(* IEC 61131-3 sources: LAxisCtrl/src/blocks, 1 file *)

(* ---- LAxisCtrl_AxisControl.st ---- *)
USING System.Math;
USING Siemens.Simatic.MotionControl.Native;

NAMESPACE Simatic.Ax.LAxisCtrl
    ///================================================================================
    /// SIEMENS AG
    /// (c)Copyright 2026 All Rights Reserved
    ///--------------------------------------------------------------------------------
    /// Library: LAxisCtrl
    /// Engineering: SIMATIC AX
    /// Restrictions: -
    /// Requirements: S7-1500T FW 4.0
    /// Functionality: This function block offers basic functionalities for axis control
    ///================================================================================
    FUNCTION_BLOCK AxisControl
        {S7.Extern = ReadWrite}
        VAR_INPUT
            /// TRUE: Enable functionality of FB
            enable : BOOL := FALSE;
            /// TRUE: Set axis enable; FALSE: Remove axis enable. MC_Power is used internally
            enableAxis : BOOL := FALSE;
            /// Rising edge: Acknowledgment of technology alarms or restart of the axis (depending on config). MC_Reset is used internally
            resetAxis : BOOL := FALSE;
            /// TRUE: Unconditionally open holding brake if axis is not enabled (e.g. for service purposes). Note: Do not modify this input while disabling of the axis is active (input enableAxis := FALSE and output axisEnabled = TRUE). MC_SetAxisSTW is used internally
            openBrake : BOOL := FALSE;
            /// Rising edge: Move an axis in jog mode (forward); Falling edge: Stop jogging. MC_MoveJog is used internally
            jogForward : BOOL := FALSE;
            /// Rising edge: Move an axis in jog mode (backward); Falling edge: Stop jogging. MC_MoveJog is used internally
            jogBackward : BOOL := FALSE;
            /// Rising edge: Move an axis at constant velocity/speed. MC_MoveVelocity is used internally
            moveVelocity : BOOL := FALSE;
            /// Rising edge: Brake an axis until it comes to a standstill. Note: MC_Halt is triggered internally
            stop : BOOL := FALSE;
            /// Rising edge: Brake an axis until it comes to a standstill (with fastStop dynamics). Note: MC_Halt is triggered internally
            fastStop : BOOL := FALSE;
            /// TRUE: Enable force/torque limiting. MC_TorqueLimiting is used internally
            torqueLimiting : BOOL := FALSE;
            /// Rising edge: Home axis. MC_Home is used internally
            homing : BOOL := FALSE;
            /// Rising edge: Move an axis relative to its position when execution of the job began. MC_MoveRelative is used internally
            posRelative : BOOL := FALSE;
            /// Rising edge: Move an axis to an absolute position. MC_MoveAbsolute is used internally
            posAbsolute : BOOL := FALSE;
            /// Rising edge: Start a superimposed positioning. MC_MoveSuperimposed is used internally
            posSuperimposed : BOOL := FALSE;
            /// Rising edge: Decelerate a superimposed motion to zero velocity. MC_HaltSuperimposed is used internally
            haltSuperimposed : BOOL := FALSE;
            /// Rising edge: Start a gearing operation (relative). MC_GearIn is used internally
            gearInRelative : BOOL := FALSE;
            /// Rising edge: Start a gearing operation (absolute). MC_GearInPos is used internally
            gearInAbsolute : BOOL := FALSE;
            /// Rising edge: Start a gearing operation (velocity synchronous). MC_GearInVelocity is used internally
            gearInVelocity : BOOL := FALSE;
            /// Rising edge: End a gearing/camming operation. MC_GearOut/MC_CamOut is used internally
            gearOutCamOut : BOOL := FALSE;
            /// Rising edge: Start a camming operation. MC_CamIn is used internally
            camIn : BOOL := FALSE;
            /// Rising edge: Start a phasing operation. MC_PhasingRelative/MC_PhasingAbsolute is used internally
            phasing : BOOL := FALSE;
            /// Rising edge: Start an offset operation. MC_OffsetRelative/MC_OffsetAbsolute is used internally
            offset : BOOL := FALSE;
            /// Reference to axis technology object to be controlled
            axis : DB_ANY  := UINT#0;
            /// Reference to leading axis technology object for synchronous motion
            master : DB_ANY := UINT#0;
            /// Cam technology object
            cam : DB_ANY := UINT#0;
            /// Structure for parameters
            config : typeAxisConfig;
        END_VAR

        {S7.Extern = ReadOnly}
        VAR_OUTPUT
            /// TRUE: Valid set of output values available at the FB
            valid : BOOL := FALSE;
            /// TRUE: FB is working and new output values can be expected
            busy : BOOL := FALSE;
            /// TRUE: An error occurred while processing the FB
            error : BOOL := FALSE;
            /// Current status of FB (16#0000 - 16#7FFF: Status of the FB, 16#8000 - 16#FFFF: Error identification)
            status : AxisStatus;
            /// Text of current status of FB
            statusText : String[STATUS_TEXT_LENGTH] := STRING#'STATUS_NO_CALL';
            /// Status of internally called subfunctions (ErrorID of Motion Control instructions)
            subfunctionStatus : WORD;
            /// TRUE: The technology object is enabled. Motion commands can be executed
            axisEnabled : BOOL := FALSE;
            /// TRUE: Reset/Restart of the axis is active
            resetActive : BOOL := FALSE;
            /// TRUE: The selected basic motion command is being executed
            commandBusy : BOOL := FALSE;
            /// TRUE: The selected basic motion command has completed without error
            commandDone : BOOL := FALSE;
            /// TRUE: The selected basic motion command has been aborted
            commandAborted : BOOL := FALSE;
            /// TRUE: The setpoint velocity/speed was reached and will be maintained
            inVelocity : BOOL := FALSE;
            /// TRUE: The drive is operating at the force/torque limit
            inLimitation : BOOL := FALSE;
            /// TRUE: Homing command is being executed
            homingCommandBusy : BOOL := FALSE;
            /// TRUE: Homing command has completed without error
            homingCommandDone : BOOL := FALSE;
            /// TRUE: Homing command has been aborted
            homingCommandAborted : BOOL := FALSE;
            /// TRUE: The selected superimposed motion command is being executed
            superimposedBusy : BOOL := FALSE;
            /// TRUE: The selected superimposed motion command  has completed without error
            superimposedDone : BOOL := FALSE;
            /// TRUE: The selected superimposed motion command has been aborted
            superimposedAborted : BOOL := FALSE;
            /// TRUE: The selected superimposed motion is active
            superimposedStart : BOOL := FALSE;
            /// TRUE: The drive is kept at the fixed stop (clamping), the axis position is within the positioning tolerance
            inClamping : BOOL := FALSE;
            /// TRUE: The axis is synchronizing to the leading axis / desynchronizing from the leading axis (Note: signal is only valid for the currently selected synchronous functionality, see outputs 'gearInAbsoluteSelected', 'gearInVelocitySelected', 'gearOutCamOutSelected' or 'camInSelected')
            startSync : BOOL := FALSE;
            /// TRUE: The axis is synchronized to the leading axis (Note: signal is only valid for the currently selected synchronous functionality, see outputs 'gearInRelativeSelected', 'gearInAbsoluteSelected', 'gearInVelocitySelected' or 'camInSelected')
            inSync : BOOL := FALSE;
            /// TRUE: The end of the cam has been reached. The output is displayed for at least one call when the cam is used cyclically
            endOfProfile : BOOL := FALSE;
            /// TRUE: Synchronous operation is being simulated
            inSimulation : BOOL := FALSE;
            /// TRUE: Jogging is active
            jogSelected : BOOL := FALSE;
            /// TRUE: Moving with constant velocity/speed is active
            moveVelocitySelected : BOOL := FALSE;
            /// TRUE: Stopping is active
            stopSelected : BOOL := FALSE;
            /// TRUE: Stopping is active (with fastStop dynamics)
            fastStopSelected : BOOL := FALSE;
            /// TRUE: Force/Torque limiting is active
            torqueLimitingSelected : BOOL := FALSE;
            /// TRUE: Homing is active
            homingSelected : BOOL := FALSE;
            /// TRUE: Relative positioning is active
            posRelativeSelected : BOOL := FALSE;
            /// TRUE: Absolute positioning is active
            posAbsoluteSelected : BOOL := FALSE;
            /// TRUE: Superimposed positioning is active (See also outputs: superimposedBusy, superimposedDone, superimposedAborted)
            posSuperimposedSelected : BOOL := FALSE;
            /// TRUE: Superimposed halting is active (See also outputs: superimposedBusy, superimposedDone, superimposedAborted)
            haltSuperimposedSelected : BOOL := FALSE;
            /// TRUE: Relative gearing is active (See also outputs: commandBusy, commandDone, commandAborted, inSync)
            gearInRelativeSelected : BOOL := FALSE;
            /// TRUE: Absolute gearing is active (See also outputs: commandBusy, commandDone, commandAborted, startSync, inSync)
            gearInAbsoluteSelected : BOOL := FALSE;
            /// TRUE: Velocity gearing is active (See also outputs: commandBusy, commandDone, commandAborted, startSync, inSync)
            gearInVelocitySelected : BOOL := FALSE;
            /// TRUE: End a gearing/camming operation is active (See also outputs: commandBusy, commandDone, commandAborted, startSync)
            gearOutCamOutSelected : BOOL := FALSE;
            /// TRUE: Camming is active (See also outputs: commandBusy, commandDone, commandAborted, startSync, inSync)
            camInSelected : BOOL := FALSE;
            /// TRUE: Phasing is active (See also outputs: superimposedBusy, superimposedDone, superimposedAborted, superimposedStart)
            phasingSelected : BOOL := FALSE;
            /// TRUE: Offset is active (See also outputs: superimposedBusy, superimposedDone, superimposedAborted, superimposedStart)
            offsetSelected : BOOL := FALSE;
            /// Diagnostics structure
            diagnostics : typeDiagnostics;
        END_VAR

        VAR
            /// Old value of statStatus
            _statusOld : AxisStatus;
            /// Internal text of current status of FB
            _statusText : String[STATUS_TEXT_LENGTH] := STRING#'STATUS_NO_CALL';
            /// Error occurred that can only be solved by user; rising edge at enable input necessary
            _errorUserCleared : BOOL := FALSE;
            /// Error occurred that can be acknowledged by FB
            _errorAutoCleared : BOOL := FALSE;
            /// Internal variable for status
            _status : AxisStatus;
            /// Internal variable for subfunction status
            _subfunctionStatus : WORD := WORD#16#0000;
            /// Internal variable for diagnostics
            _diagnostics : typeDiagnostics;
            /// Old value of enable for edge detection
            _enableOld : BOOL := FALSE;
            /// State of FB (function block state machine)
            _state : SINT := AXIS_MOTION;
            /// TRUE: First cycle of reset command
            _firstCycleReset : BOOL := TRUE;
            /// Old value of MC_Power.error
            _powerErrorOld : BOOL := FALSE;
            /// State of reset command
            _resetState : INT := CMD_IDLE;
            /// TRUE: First cycle of error in reset command
            _firstCycleResetError : BOOL := FALSE;
            /// Variable for requested extended command (e.g. resetAxis, torquelimiting, homing)
            _extendedCommand : DWORD := CMD_NO_SELECTION;
            /// Old value of variable for requested extended command
            _extendedCommandOld : DWORD := CMD_NO_SELECTION;
            /// Old value of enableAxis for edge detection
            _enableAxisOld : BOOL := FALSE;
            /// Internal empty diagnostic structure
            _emptyDiagnostics : typeDiagnostics;
            /// Old value of variable for homing command input
            _homingOld : BOOL := FALSE;
            /// TRUE: First cycle in homing command
            _firstCycleHoming : BOOL := TRUE;
            /// Current selected passive homing mode
            _passiveHomingState : DINT := NO_HOMING_ACTIVE;
            /// Current state of execution of homing command
            _exeOfHoming : INT := CMD_BUSY;
            /// Variable for requested basic motion command
            _basicCommand : DWORD := CMD_NO_SELECTION;
            /// Old value of variable for requested basic motion command
            _basicCommandOld : DWORD := CMD_NO_SELECTION;
            /// State of selected basic motion command
            _basicMotionState : DINT := NO_SELECTION;
            /// State of execution of current state of basic motion
            _exeOfBasicMotion : INT := CMD_BUSY;
            /// TRUE: First cycle in respective state for basic motion functionality
            _firstCycleBasicMotion : BOOL := TRUE;
            /// TRUE: applicative error occurred (e.g. invalid direction configured)
            _applicativeBasicMotionError : BOOL := FALSE;
            /// Velocity change on the fly is active
            _velocityChangeOnTheFly : BOOL := FALSE;
            /// Internal variable for velocity
            _basicVelocity : LREAL := 0.0;
            /// Internal variable for acceleration
            _basicAcceleration : LREAL := 0.0;
            /// Internal variable for deceleration
            _basicDeceleration : LREAL := 0.0;
            /// Internal variable for jerk
            _basicJerk : LREAL := 0.0;
            /// TRUE: First cycle of done at fastStop
            _firstCycleDone : BOOL := FALSE;
            /// Current executed state for torquelimiting functionality
            _torqueLimitingState : SINT := NO_TORQUE_LIMITING_ACTIVE;
            /// TRUE: Error at Torquelimiting occurred last cycle
            _torqueLimitingErrorOld : BOOL := FALSE;
            /// Current selected jog mode
            _jogMode : DINT := JOG_MODE_CONTINUOUS;
            /// Internal variable for direction of rotation of the axis
            _direction : INT := SPECIFIED_DIR;
            /// Internal variable for stopOnError function
            _stopWithoutSignalization : BOOL;
            /// Brake is opened
            _brakeOpened : BOOL;
            /// Brake change active
            _brakeChangeActive : BOOL;
            /// Edge detection
            _openBrakeOld : BOOL;
            /// The specified value is used according to the selected "Mode".
            _homingPosition : LREAL := 0.0;
            /// Current subState of execution of homing functionality
            _homingSubState : SINT := HOMING_IDLE;
            /// Current subState of execution of jog incremental functionality
            _incJogSubState : SINT := INC_JOG_IDLE;
            /// Last stored axis position (for incremental jogging)
            _incJogStartPosition : LREAL := 0.0;
            /// Old value of direction of executing incremental jogging
            _incJogDirectionOld : INT := 0;
            /// Jog Incremental: distance of Increment (positive or negative)
            _increment : LREAL := 0.0;
            /// Jog Incremental: current distance to destination position
            _incJogDistance : LREAL := 0.0;
            /// TRUE: First cycle in incremental jogging state (detection of new increment)
            _resetIncJog : BOOL := TRUE;
            /// Internal variable for position
            _position : LREAL := 0.0;
            /// Position change on the fly is active
            _positionChangeOnTheFly : BOOL := FALSE;
            /// Current selected active homing mode
            _activeHomingState : DINT := NO_HOMING_ACTIVE;
            /// Variable for requested superimposed motion command
            _supImpCommand : DWORD := CMD_NO_SELECTION;
            /// Old value of variable for requested superimposed motion command
            _supImpCommandOld : DWORD := CMD_NO_SELECTION;
            /// Current selected superimposed motion functionality
            _supImpMotionState : DINT := NO_SELECTION;
            /// Current state of execution of superimposed basic motion
            _exeOfSupImpMotionState : INT := CMD_BUSY;
            /// TRUE: First cycle in positioning (superimposed) functionality
            _firstCycleSupImpMotion : BOOL := TRUE;
            /// Position setpoint (for posSuperimposed command)
            _supImpMotionPosition : LREAL := 0.0;
            /// TRUE: applicative error occurred (e.g. invalid direction configured)
            _applicativeSupImpMotionError : BOOL := FALSE;
            /// Ratio change on the fly is active
            _ratioChangeOnTheFly : BOOL := FALSE;
            /// Gear ratio numerator
            _ratioNumerator : DINT := 1;
            /// Gear ratio denominator
            _ratioDenominator : DINT := 1;
            /// Phase shift change on the fly is active
            _changePhaseShiftOnTheFly : BOOL := FALSE;
            /// Offset change on the fly is active
            _changeOffsetOnTheFly : BOOL := FALSE;
            /// Relative/Absolute master value shift
            _phaseShift : LREAL := 0.0;
            /// Indicates the type of phase shift (TRUE: The phase shift is taken over as an absolute value; FALSE: The phase shift is added to an existing offset)
            _phaseAbsolute : BOOL := TRUE;
            /// Indicates the type of offset shift (TRUE: The offset shift is taken over as an absolute value; FALSE: The offset shift is added to an existing offset)
            _offsetAbsolute : BOOL := FALSE;
            /// Relative/Absolute offset
            _offsetValue : LREAL := 0.0;
            /// Type of axis
            _typeAxis : INT;
            /// Internal variable for enabling axis
            _enableAxis : BOOL := FALSE;
            /// Current executed state for synchronized motion simulation
            _syncMotionSimulationState : SINT := AXIS_NOT_IN_SIM;
            /// Old value of MC_SynchronizedMotionSimulation.error
            _synchronizedMotionErrorOld : BOOL := FALSE;
            /// Current executed State for execution of basic motion commands or reset of waiting gearing / camming commands
            _mainSelectionState : INT := 0;
            /// Application of cam
            _applicationMode : DINT := 0;
            /// Internal variable for waiting function state
            _waitingFunctionState : DINT := 0;
            /// Internal variable for waiting function state
            _waitingFunctionStateAbortAutomatic : DINT := -1;
            /// Internal variable for function state
            _functionState : DINT := 0;
            /// Internal variable
            _gearAndCamOutMode : DINT := 0;
            /// Internal variable
            _syncOutState : DINT;
            /// Internal old value for cam
            _camOld : DB_ANY;
            /// Internal old value for master
            _masterOld : DB_ANY;
            /// Internal reference of the technology object type TO_CamBase
            _refCamBase : REF_TO TO_CamBase;
            /// Internal reference of the technology object type TO_Axis (for the master axis)
            _refMasterAxis : REF_TO TO_Axis;
            /// Internal reference of the technology object type TO_Axis
            _refAxis : REF_TO TO_Axis;
            /// Internal reference of the technology object type TO_ExternalEncoder
            _refExtEncoder : REF_TO TO_ExternalEncoder;
            /// Internal reference of the technology object type TO_SpeedAxis
            _refSpeedAxis : REF_TO TO_SpeedAxis;
            /// Internal reference of the technology object type TO_PositioningAxis
            _refPosAxis : REF_TO TO_PositioningAxis;
            /// Internal reference of the technology object type TO_SynchronousAxis
            _refSyncAxis : REF_TO TO_SynchronousAxis;
            /// Instance of MC_Power
            _instPower : MC_POWER;
            /// Instance of MC_Reset
            _instReset : MC_RESET;
            /// Instance of MC_Home
            _instHome : MC_HOME;
            /// Instance of MC_Halt
            _instHalt : MC_HALT;
            /// Instance of MC_MoveJog
            _instMoveJog : MC_MOVEJOG;
            /// Instance of MC_TorqueLimiting
            _instTorqueLimiting : MC_TORQUELIMITING;
            /// Instance of MC_MoveVelocity
            _instMoveVelocity : MC_MOVEVELOCITY;
            /// Instance of MC_SetAxisSTW
            _instSetAxisSTW : MC_SETAXISSTW;
            /// Instance of MC_MoveRelative
            _instMoveRelative : MC_MOVERELATIVE;
            /// Instance of MC_MoveAbsolute
            _instMoveAbsolute : MC_MOVEABSOLUTE;
            /// Instance of MC_MoveSuperimposed
            _instMoveSuperimposed : MC_MOVESUPERIMPOSED;
            /// Instance of MC_HaltSuperimposed
            _instHaltSuperimposed : MC_HALTSUPERIMPOSED;
            /// Instance of MC_GearIn
            _instGearIn : MC_GEARIN;
            /// Instance of MC_PhasingAbsolute
            _instPhasingAbsolute : MC_PHASINGABSOLUTE;
            /// Instance of MC_PhasingRelative
            _instPhasingRelative : MC_PHASINGRELATIVE;
            /// Instance of MC_OffsetAbsolute
            _instOffsetAbsolute : MC_OFFSETABSOLUTE;
            /// Instance of MC_OffsetRelative
            _instOffsetRelative : MC_OFFSETRELATIVE;
            /// Instance of MC_GearInPos
            _instGearInPos : MC_GEARINPOS;
            /// Instance of MC_GearInVelocity
            _instGearInVelocity : MC_GEARINVELOCITY;
            /// Instance of MC_GearOut
            _instGearOut : MC_GEAROUT;
            /// Instance of MC_CamIn
            _instCamIn : MC_CAMIN;
            /// Instance of MC_CamOut
            _instCamOut : MC_CAMOUT;
            /// Instance of MC_SynchronizedMotionSimulation
            _instSyncMotionSimulation : MC_SYNCHRONIZEDMOTIONSIMULATION;
        END_VAR

        VAR_TEMP
            // Temporary variable for enable FB
            tempEnable : BOOL;
            // Temporary variable for extended command
            tempNewExtendedCmd : DINT;
            // Temporary variable for enableAxis
            tempEnableAxis : BOOL;
            // Temporary variable for error in actual command
            tempErrorInCmd : BOOL;
            // Temporary DWord which indicates all rising edges of command word
            tempRisingCmd : DWORD;
            // TRUE: Stop or faststop selected in current cycle
            tempStopCmdSelected : BOOL;
            // Temporary variable for statusword of axis
            tempStatusWord : DWORD;
            // Temporary variable for open brake
            tempOpenBrake : BOOL;
            // Temporary DWord for evaluation of rising edges of basic command word
            tempDword : DWORD;
            // Temporary index
            tempIndex : INT;
            // Temporary counter for rising edges in command word
            tempCountRisEdges : USINT;
            // Temporary variable for basic motion command
            tempNewBasicMotionCmd : DINT;
            // TRUE: State change is active, stay in loop for one more cycle
            tempStateChangeActive : BOOL;
            // Temporary variable for superimposed motion command
            tempNewSupImpCmd : DINT;
            // Temporary DInt variable
            tempDInt : DINT;
            // Temporary LReal variable
            tempLReal : LREAL;
            // Temporary Bool variable
            tempBool : BOOL;
            // Temporary variable for homing command
            tempHoming : BOOL;
        END_VAR

        VAR CONSTANT
            // Axis type: External encoder
            EXTERNAL_ENCODER : INT := 1;
            // Axis type: Speed axis
            SPEED_AXIS : INT := 2;
            // Axis type: Positioning axis
            POS_AXIS : INT := 3;
            // Axis type: Synchronous axis
            SYNC_AXIS : INT := 4;
            // Length of status text
            STATUS_TEXT_LENGTH : INT := 39;
            // State of FB: MotionState, new commands are evaluated
            AXIS_MOTION : SINT := SINT#1;
            // State of FB: Error, falling edge at FB_ENABLE required
            FB_ERROR : SINT := SINT#5;
            // No command is selected
            CMD_NO_SELECTION : DWORD := DWORD#16#0000_0000;
            // State of basicMotion/superimposedMotion: No execution of a command
            NO_SELECTION : INT := 0;

            // State of FB: StoppingState, MC_HALT is executed, new commands are not evaluated
            AXIS_FAST_STOPPING : SINT := SINT#2;
            // State of FB: ErrorState: Selection if StopOnError must be executed (depending on config)
            AXIS_STOP_ON_ERROR_SELECTION : SINT := SINT#3;
            // State of FB: ErrorState: Execution of StopOnError
            AXIS_STOP_ON_ERROR_EXECUTION : SINT := SINT#4;

            // Jogmode continuous selected (MC_MOVEJOG)
            JOG_MODE_CONTINUOUS : INT := 0;

            // State of basicMotion: Execution of fast stop command
            FAST_STOP_SELECTED : INT := 1;
            // State of basicMotion: Execution of stop command
            STOP_SELECTED : INT := 2;
            // State of basicMotion: Execution of jog forward command
            JOG_FORWARD_SELECTED : INT := 4;
            // State of basicMotion: Execution of jog backward command
            JOG_BACKWARD_SELECTED : INT := 8;
            // State of basicMotion: Execution of jog command if forward and backward are selected
            JOG_FW_AND_BW_SELECTED : INT := 12;
            // State of basicMotion: Execution of move velocity command
            MOVE_VELOCITY_SELECTED : INT := 16;
            // State of basicMotion: Execution of active homing command
            ACTIVE_HOMING_SELECTED : INT := 1024;
            // State of basicMotion: Execution of position command (relative)
            POS_RELATIVE_SELECTED : INT := 32;
            // State of basicMotion: Execution of position command (absolute)
            POS_ABSOLUTE_SELECTED : INT := 64;
            // State of basicMotion: Execution of gearIn command
            GEAR_IN_RELATIVE_SELECTED : INT := 128;
            // State of basicMotion: Execution of gearInPos command
            GEAR_IN_ABSOLUTE_SELECTED : INT := 256;
            // State of basicMotion: Execution of gearInVelocity command
            GEAR_IN_VELOCITY_SELECTED : INT := 4096;
            // State of basicMotion: Execution of camIn command
            CAM_IN_SELECTED : INT := 512;
            // State of basicMotion: Execution of gear and camOut command
            GEAR_OUT_CAM_OUT_SELECTED : INT := 2048;
            // State of superimposedMotion: Execution of posSuperimposed command
            POS_SUPERIMPOSED_SELECTED : INT := 1;
            // State of superimposedMotion: Execution of haltSuperimposed command
            HALT_SUPERIMPOSED_SELECTED : INT := 8;
            // State of superimposedMotion: Execution of phasing command
            PHASING_SELECTED : INT := 2;
            // State of superimposedMotion: Execution of offset command
            OFFSET_SELECTED : INT := 4;

            // State of basicMotion command: No execution
            CMD_IDLE : INT := 0;
            // State of basicMotion command: Subsequent call
            CMD_BUSY : INT := 1;
            // State of basicMotion command: Finished with "DONE"
            CMD_DONE : INT := 2;
            // State of basicMotion command: Finished with "ABORTED"
            CMD_ABORTED : INT := 4;
            // State of basicMotion command: Finished with "ERROR"
            CMD_ERROR : INT := 8;
            // State of basicMotion command: Finished with other reason
            CMD_END_PROCESS : INT := 16;

            // State of torquelimiting command: Not enabled
            NO_TORQUE_LIMITING_ACTIVE : SINT := SINT#0;
            // State of torquelimiting command: Torquelimiting is active
            TORQUE_LIMITING_SELECTED : SINT := SINT#1;
            // State of torquelimiting command: Torquelimiting is disabling
            TORQUE_LIMITING_DISABLE : SINT := SINT#10;

            // First bitposition for detecting rising edges at basic motion command word
            BITPOSITION_BASIC_MOTION_CMD : SINT := SINT#4;
            // Last bitposition for detecting rising edges at command word
            BIT_POS_LAST : SINT := SINT#15;
            // The sign of the velocity specified at the "Velocity" parameter defines the direction of rotation.
            SPECIFIED_DIR : INT := 0;
            // Bit 12 in STW
            MASK_STW_BIT12 : WORD := WORD#16#1000;

            // State of homing command: No homing active
            NO_HOMING_ACTIVE : SINT := SINT#-10;
            // State of homing command: (Standard) homing with MC_HOME
            STANDARD_HOMING : SINT := SINT#-1;

            // First bitposition for detecting rising edges at superimposed motion command word
            BITPOSITION_SUPERIMPOSED_MOTION_CMD : SINT := SINT#0;

            // State of torquelimiting command: Homing on fixed stop is active
            FIXED_STOP_DETECTION_ACTIVE : SINT := SINT#2;
            // State of torquelimiting command: Homing on fixed stop is finished
            FIXED_STOP_DETECTION_FINISHED : SINT := SINT#3;
            // State of torquelimiting command: Error occurred at homing on fixed stop process, axis is in clamping
            FIXED_STOP_DETECTION_ERROR_IN_CLAMPING : SINT := SINT#5;
            // State of torquelimiting command: Error occurred at homing on fixed stop process, axis is not in clamping
            FIXED_STOP_DETECTION_ERROR_NOT_IN_CLAMPING : SINT := SINT#6;

            // State of homing command: Applicative homing on fixed stop process active
            HOMING_ON_FIXED_STOP : SINT := SINT#0;
            // State of homing command: Applicative homing on fixed stop with moving out of clamping process active
            HOMING_ON_FIXED_STOP_WITH_MOVING_OUT_OF_CLAMPING : SINT := SINT#1;
            // State of homing command: Applicative homing on fixed stop with moving to target position process active
            HOMING_ON_FIXED_STOP_WITH_MOVING_TO_TARGET_POSITION : SINT := SINT#2;

            // Scaling factor for moving out of clamping. 1.0 = positioning window
            DISTANCE_SCALING : LREAL := 1.05;
            // Fixed stop detection (Mode for MC_TORQUELIMITING)
            MODE_FIXED_STOP_DETECTION : INT := 1;
            // Positive/Forward direction of rotation
            FORWARD_DIR : INT := 1;
            // Negative/Backward direction of rotation
            BACKWARD_DIR : INT := 2;
            // Shortest path
            SHORTEST_WAY_DIR : INT := 3;
            // Direct homing (absolute). Parameter "position" at MC_HOME is effective
            DIRECT_HOMING : INT := 0;
            // Active homing. Parameter "position" at MC_HOME is effective
            ACTIVE_HOMING : INT := 3;
            // Active homing. The configured home position value in technology object is effective
            ACTIVE_HOMING_TO_DEF_VALUE : INT := 5;
            // Absolute encoder adjustment (absolute)
            ABSOLUTE_ENCODER_ADJUSTMENT : INT := 7;
            // Encodertype INCREMENTAL
            INCREMENTAL_ENCODER : INT := 0;

            // SubState of homing on fixed stop process: Idle
            HOMING_IDLE : SINT := SINT#0;
            // SubState of homing on fixed stop process: Detecting fixed stop
            HOMING_FIXED_STOP_DETECTION : SINT := SINT#1;
            // SubState of homing on fixed stop process: Homeprocess (MC_HOME)
            HOMING_PROCESS : SINT := SINT#2;
            // SubState of homing on fixed stop process: Positioning to homeposition
            HOMING_POSITION : SINT := SINT#3;

            // Substate of incremental jog process: Idle
            INC_JOG_IDLE : SINT := SINT#0;
            // Substate of incremental jog process: Start moving
            INC_JOG_START : SINT := SINT#1;
            // Substate of incremental jog process: Stop moving
            INC_JOG_STOP : SINT := SINT#3;

            // Jogmode incremental selected - start always with new increment when command is selected
            JOG_MODE_NEW_INCREMENT : INT := 1;
            // Jogmode incremental selected - continue with increment when command is selected again
            JOG_MODE_CONTINUE_INCREMENT : INT := 2;
            // Application of the cam: Once/not cyclic (MC_CAMIN)
            APPLICATION_MODE_ONCE : INT := 0;
            // State of MainSelectionState: Regular execution of basic motion commands
            CALL_BASIC_MOTION : INT := 0;
            // State of MainSelectionState: Reset of waiting synchronous commands
            ABORT_WAITING_GEARINPOS_OR_CAMIN : INT := 1;

            // Mode for MC_GearOut / MC_CamOut instruction
            CANCEL_ONLY_WAITING_GEARING_CAMMING : DINT := 5;
            // No operation active or waiting
            WFS_FS_NO_OPERATION : DINT := 0;
            // Function state / Waiting function state: GearIn
            WFS_FS_GEARIN : DINT := 1;
            // Function state / Waiting function state: GearInPos
            WFS_FS_GEARINPOS : DINT := 2;
            // Function state / Waiting function state: CamIn
            WFS_FS_CAMIN : DINT := 3;
            // Function state / Waiting function state: Gearout
            WFS_FS_GEAROUT : DINT := 4;
            // Function state / Waiting function state: CamOut
            WFS_FS_CAMOUT : DINT := 5;

            // GearOutCamOut mode: Automatic
            SYNCOUT_MODE_AUTOMATIC : DINT := -1;
            // GearOutCamOut mode: GearOut
            SYNCOUT_MODE_GEAROUT : DINT := 0;
            // GearOutCamOut mode: CamOut
            SYNCOUT_MODE_CAMOUT : DINT := 1;
            // Sync out state
            SYNCOUT_STATE_CHECK_WAITING : INT := 1;
            // Sync out state
            SYNCOUT_STATE_GEAROUT_WAITING_BUSY : INT := 2;
            // Sync out state
            SYNCOUT_STATE_CAMOUT_WAITING_BUSY : INT := 3;
            // Sync out state
            SYNCOUT_STATE_CHECK_ACTIVE : INT := 4;
            // Sync out state
            SYNCOUT_STATE_GEAROUT_ACTIVE_BUSY : INT := 5;
            // Sync out state
            SYNCOUT_STATE_CAMOUT_ACTIVE_BUSY : INT := 6;
            // Sync out state
            SYNCOUT_STATE_DONE : INT := 7;
            // Sync out state
            SYNCOUT_STATE_ABORTED : INT := 8;
            // Sync out state
            SYNCOUT_STATE_ERROR : INT := 9;

            // State of motionSimulation: Axis is not in simulation
            AXIS_NOT_IN_SIM : SINT := SINT#0;
            // State of motionSimulation: Setting axis in simulation
            AXIS_STATE_SET_SIM : SINT := SINT#1;
            // State of motionSimulation: Disable axis
            AXIS_DISABLE : SINT := SINT#2;
            // State of motionSimulation: Axis is in simulation
            AXIS_STATE_IN_SIM : SINT := SINT#3;
            // State of motionSimulation: Enable axis
            AXIS_ENABLE : SINT := SINT#4;
            // State of motionSimulation: Resetting axis simulation
            AXIS_STATE_RESET_SIM : SINT := SINT#5;
        END_VAR

        //----------------------------------------------------------------------------------------------
        // Enable / disable FB
        //----------------------------------------------------------------------------------------------
        tempEnable := enable; // Create temporary process image
        IF NOT tempEnable AND _enableOld THEN

            // Reset outputs
            // ==========================================================
            // Error and valid outputs are reset with falling edge of enable input
            error := FALSE;
            valid := FALSE;
            status := AxisStatus#STATUS_NO_CALL;
            statusText := STRING#'STATUS_NO_CALL';
            subfunctionStatus := WORD#16#0000;
            _subfunctionStatus := WORD#16#0000;

            // Reset status outputs
            axisEnabled := FALSE;
            resetActive := FALSE;

            // Reset outputs for homing commands
            homingCommandBusy := FALSE;
            homingCommandDone := FALSE;
            homingCommandAborted := FALSE;
            homingSelected := FALSE;
            // Reset outputs for torquelimiting command
            torqueLimitingSelected := FALSE;
            inLimitation := FALSE;

            // Reset outputs for basic motion commands
            commandDone := FALSE;
            commandBusy := FALSE;
            commandAborted := FALSE;
            inVelocity := FALSE;
            fastStopSelected := FALSE;
            stopSelected := FALSE;
            jogSelected := FALSE;
            moveVelocitySelected := FALSE;
            // Outputs for for up to LAxisCtrl_PosAxis
            posRelativeSelected := FALSE;
            posAbsoluteSelected := FALSE;
            inClamping := FALSE;

            // Reset outputs for superimposed motion commands
            superimposedBusy := FALSE;
            superimposedDone := FALSE;
            superimposedAborted := FALSE;
            superimposedStart := FALSE;
            posSuperimposedSelected := FALSE;
            haltSuperimposedSelected := FALSE;
            startSync := FALSE;
            inSync := FALSE;
            endOfProfile := FALSE;
            gearInRelativeSelected := FALSE;
            inSimulation := FALSE;
            gearInAbsoluteSelected := FALSE;
            gearInVelocitySelected := FALSE;
            phasingSelected := FALSE;
            offsetSelected := FALSE;
            camInSelected := FALSE;
            gearOutCamOutSelected := FALSE;

            // Reset internal variables
            // ==========================================================
            _errorUserCleared := FALSE;
            _errorAutoCleared := FALSE;
            _status := AxisStatus#STATUS_NO_CALL;
            _statusOld := AxisStatus#STATUS_NO_CALL;
            _diagnostics := _emptyDiagnostics;

            _state := AXIS_MOTION;
            _firstCycleReset := FALSE;
            _powerErrorOld := FALSE;
            _resetState := CMD_IDLE;
            _firstCycleResetError := FALSE;

            _extendedCommand := CMD_NO_SELECTION;
            _extendedCommandOld := CMD_NO_SELECTION;
            _enableAxisOld := FALSE;
            _homingOld := FALSE;
            _firstCycleHoming := FALSE;
            _passiveHomingState := NO_HOMING_ACTIVE;
            _exeOfHoming := CMD_BUSY;
            _basicCommand := CMD_NO_SELECTION;
            _basicCommandOld := CMD_NO_SELECTION;
            _basicMotionState := NO_SELECTION;
            _exeOfBasicMotion := CMD_BUSY;
            _firstCycleBasicMotion := FALSE;
            _applicativeBasicMotionError := FALSE;
            _velocityChangeOnTheFly := FALSE;
            _basicVelocity := 0.0;
            _basicAcceleration := 0.0;
            _basicDeceleration := 0.0;
            _basicJerk := 0.0;

            _firstCycleDone := FALSE;

            _torqueLimitingState := NO_TORQUE_LIMITING_ACTIVE;
            _torqueLimitingErrorOld := FALSE;
            _jogMode := JOG_MODE_CONTINUOUS;
            _direction := SPECIFIED_DIR;

            _homingPosition := 0.0;
            _homingSubState := HOMING_IDLE;
            _incJogSubState := INC_JOG_IDLE;
            _incJogStartPosition := 0.0;
            _incJogDirectionOld := 0;
            _increment := 0.0;
            _incJogDistance := 0.0;
            _resetIncJog := TRUE;
            _position := 0.0;
            _positionChangeOnTheFly := FALSE;

            _activeHomingState := NO_HOMING_ACTIVE;
            _supImpCommand := CMD_NO_SELECTION;
            _supImpCommandOld := CMD_NO_SELECTION;
            _supImpMotionState := NO_SELECTION;
            _exeOfSupImpMotionState := CMD_BUSY;
            _firstCycleSupImpMotion := FALSE;
            _supImpMotionPosition := 0.0;
            _applicativeSupImpMotionError := FALSE;
            _ratioChangeOnTheFly := FALSE;
            _ratioNumerator := 0;
            _ratioDenominator := 0;
            // Tags for synchronized motion simulation
            _changePhaseShiftOnTheFly := FALSE;
            _changeOffsetOnTheFly := FALSE;
            _phaseShift := 0.0;
            _offsetValue := 0.0;
            _phaseAbsolute := TRUE;
            _offsetAbsolute := TRUE;
            _enableAxis := FALSE;
            _syncMotionSimulationState := AXIS_NOT_IN_SIM;
            _synchronizedMotionErrorOld := FALSE;
            _mainSelectionState := 0;
            _applicationMode := 0;

            _waitingFunctionState := 0;
            _waitingFunctionStateAbortAutomatic := -1;
            _functionState := 0;
            // ===========================================================

            // Disable Axis
            IF (_instPower.Busy = TRUE) THEN
                _instPower(Axis := _refAxis^,
                           Enable := FALSE,
                           StartMode := config.power.startMode,
                           StopMode := config.power.stopMode);
                // Check if error occurred
                IF (_instPower.Error = TRUE) THEN
                    // Write only diagnostics if error occurred at falling edge of MC_POWER
                    diagnostics.status := AxisStatus#ERR_MC_POWER;
                    diagnostics.subfunctionStatus := _instPower.ErrorId;
                    diagnostics.basicMotionState := _basicMotionState;
                    diagnostics.superimposedMotionState := _supImpMotionState;
                END_IF;
            END_IF;

            // Reset old values for master and cam
            _masterOld := UINT#0;
            _camOld := UINT#0;

            // Set axis references to null when block is being disabled
            _refAxis := NULL;
            _refSpeedAxis := NULL;
            _refPosAxis := NULL;
            _refSyncAxis := NULL;
            _refExtEncoder := NULL;
            _refMasterAxis := NULL;
            _refCamBase := NULL;

            // Set old value of enable for edge detection and end execution
            _enableOld := tempEnable;
            RETURN;

        // Check if FB is enabled - first cycle
        ELSIF tempEnable AND NOT _enableOld THEN

            // Busy is set at rising edge of enable input
            busy := TRUE;
            status := AxisStatus#STATUS_FB_FIRST_CALL;
            statusText := STRING#'STATUS_FB_FIRST_CALL';
            // StatStatus will be written in next cycle
            _status := AxisStatus#STATUS_SUBSEQUENT_CALL;
            _statusText := STRING#'STATUS_SUBSEQUENT_CALL';

            // Reset error and diagnostics outputs
            _errorUserCleared := FALSE;
            _errorAutoCleared := FALSE;
            diagnostics := _emptyDiagnostics;
            _diagnostics := _emptyDiagnostics;

            // Copy inputs
            _extendedCommand.%X0 := resetAxis;
            _basicCommand.%X8 := gearInAbsolute;
            _basicCommand.%X12 := gearInVelocity;
            _basicCommand.%X9 := camIn;
            _basicCommand.%X11 := gearOutCamOut;
            _supImpCommand.%X1 := phasing;
            _supImpCommand.%X2 := offset;
            _basicCommand.%X7 := gearInRelative;
            _basicCommand.%X5 := posRelative;
            _basicCommand.%X6 := posAbsolute;
            _supImpCommand.%X0 := posSuperimposed;
            _supImpCommand.%X3 := haltSuperimposed;
            _supImpCommandOld := _supImpCommand;

            _basicCommand.%X0 := fastStop;
            _basicCommand.%X1 := stop;
            _basicCommand.%X2 := jogForward;
            _basicCommand.%X3 := jogBackward;
            _basicCommand.%X4 := moveVelocity;
            _basicCommandOld := _basicCommand;
            // Set old value of homing input
            _homingOld := homing;

            _extendedCommandOld := _extendedCommand;
            // Set old value of enable for edge detection and end execution
            _enableOld := tempEnable;

            // resolve reference for axis input as TO_Axis (basic type for all axes)
            _refAxis := AsAxisRef(axis);
            IF _refAxis = NULL THEN
                // Invalid axis
                error := TRUE;
                _errorUserCleared := TRUE;
                status := AxisStatus#ERR_INVALID_AXIS;
                statusText := STRING#'ERR_INVALID_AXIS';
                diagnostics.status := AxisStatus#ERR_INVALID_AXIS;
            END_IF;

            CASE GetType(axis) OF
                TO_Type#SynchronousAxis:
                    _typeAxis := SYNC_AXIS;

                    // attempt to resolve all inherited technology objects (TO_SpeedAxis, TO_PositioningAxis, TO_SynchronousAxis)
                    _refSpeedAxis := AsSpeedAxisRef(axis);
                    _refPosAxis := AsPositioningAxisRef(axis);
                    _refSyncAxis := AsSynchronousAxisRef(axis);

                    // TODO: generate other error for this case?
                    IF _refSpeedAxis = NULL OR _refPosAxis = NULL OR _refSyncAxis = NULL THEN
                        // Invalid axis
                        error := TRUE;
                        _errorUserCleared := TRUE;
                        status := AxisStatus#ERR_INVALID_AXIS;
                        statusText := STRING#'ERR_INVALID_AXIS';
                        diagnostics.status := AxisStatus#ERR_INVALID_AXIS;
                    END_IF;

                TO_Type#PositioningAxis:
                    _typeAxis := POS_AXIS;

                    // attempt to resolve all inherited technology objects (TO_SpeedAxis, TO_PositioningAxis)
                    _refSpeedAxis := AsSpeedAxisRef(axis);
                    _refPosAxis := AsPositioningAxisRef(axis);

                    // TODO: generate other error for this case?
                    IF _refSpeedAxis = NULL OR _refPosAxis = NULL THEN
                        // Invalid axis
                        error := TRUE;
                        _errorUserCleared := TRUE;
                        status := AxisStatus#ERR_INVALID_AXIS;
                        statusText := STRING#'ERR_INVALID_AXIS';
                        diagnostics.status := AxisStatus#ERR_INVALID_AXIS;
                    END_IF;

                TO_Type#SpeedAxis:
                    _typeAxis := SPEED_AXIS;

                    _refSpeedAxis := AsSpeedAxisRef(axis);

                    // TODO: generate other error for this case?
                    IF _refSpeedAxis = NULL THEN
                        // Invalid axis
                        error := TRUE;
                        _errorUserCleared := TRUE;
                        status := AxisStatus#ERR_INVALID_AXIS;
                        statusText := STRING#'ERR_INVALID_AXIS';
                        diagnostics.status := AxisStatus#ERR_INVALID_AXIS;
                    END_IF;

                TO_Type#ExternalEncoder:
                    _typeAxis := EXTERNAL_ENCODER;

                    _refExtEncoder := AsExternalEncoderRef(axis);

                    // TODO: generate other error for this case?
                    IF _refExtEncoder = NULL THEN
                        // Invalid axis
                        error := TRUE;
                        _errorUserCleared := TRUE;
                        status := AxisStatus#ERR_INVALID_AXIS;
                        statusText := STRING#'ERR_INVALID_AXIS';
                        diagnostics.status := AxisStatus#ERR_INVALID_AXIS;
                    END_IF;

                ELSE
                    // Invalid axis
                    error := TRUE;
                    _errorUserCleared := TRUE;
                    status := AxisStatus#ERR_INVALID_AXIS;
                    statusText := STRING#'ERR_INVALID_AXIS';
                    diagnostics.status := AxisStatus#ERR_INVALID_AXIS;
            END_CASE;
        RETURN;

        // Check if function block is disabled or UserClearedError is present
        ELSIF NOT tempEnable OR _errorUserCleared THEN

            IF (tempEnable = FALSE) THEN
                status := AxisStatus#STATUS_NO_CALL;
                statusText := STRING#'STATUS_NO_CALL';
            END_IF;

            // Disable Axis
            IF (_instPower.Busy = TRUE) THEN
                _instPower(Axis := _refAxis^,
                           Enable := FALSE,
                           StartMode := config.power.startMode,
                           StopMode := config.power.stopMode);
                // Check if error occurred
                IF (_instPower.Error = TRUE) THEN
                    diagnostics.status := AxisStatus#ERR_MC_POWER;
                    diagnostics.subfunctionStatus := _instPower.ErrorId;
                    diagnostics.basicMotionState := _basicMotionState;
                    diagnostics.superimposedMotionState := _supImpMotionState;
                END_IF;
            ELSE
                // Reset if torque limiting is busy and axis is disabled
                IF (_instTorqueLimiting.Busy = TRUE)
                    OR (_instSyncMotionSimulation.Busy = TRUE)
                THEN
                    _instTorqueLimiting(Axis := _refSpeedAxis^,
                                        Enable := FALSE);
                    // Disable synchronized motion simulation
                    _instSyncMotionSimulation(Slave := _refSyncAxis^,
                                              Enable := FALSE);
                ELSE
                    busy := FALSE;
                END_IF;
            END_IF;

            // Reset old values for master and cam
            _masterOld := UINT#0;
            _camOld := UINT#0;

            // Set axis references to null when block is being disabled
            _refAxis := NULL;
            _refSpeedAxis := NULL;
            _refPosAxis := NULL;
            _refSyncAxis := NULL;
            _refExtEncoder := NULL;
            _refMasterAxis := NULL;
            _refCamBase := NULL;

            _enableOld := tempEnable;
            RETURN;

        ELSE

            // Read status word of the axis cyclically (needed for MC_Power call)
            CASE _typeAxis OF // Axis type is determined (checked) when the FB is enabled
                SPEED_AXIS, POS_AXIS, SYNC_AXIS:
                    // Axis type is TO_SpeedAxis or TO_PositioningAxis or TO_SynchronousAxis
                    tempStatusWord := _refSpeedAxis^.StatusWord;

                EXTERNAL_ENCODER:
                    // Axis type is TO_ExternalEncoder
                    tempStatusWord := _refExtEncoder^.StatusWord;

                ELSE
                    // Invalid axis
                    tempStatusWord := DWORD#16#0000_0000;
            END_CASE;

            // Copy extended inputs
            _extendedCommand.%X0 := resetAxis;
            tempEnableAxis := enableAxis;
            _extendedCommand.%X1 := torqueLimiting;
            _basicCommand.%X0 := fastStop;
            _basicCommand.%X1 := stop;
            _basicCommand.%X2 := jogForward;
            _basicCommand.%X3 := jogBackward;
            _basicCommand.%X4 := moveVelocity;
            tempOpenBrake := openBrake;
            _basicCommand.%X5 := posRelative;
            _basicCommand.%X6 := posAbsolute;
            _supImpCommand.%X0 := posSuperimposed;
            _supImpCommand.%X3 := haltSuperimposed;
            tempHoming := homing;
            IF (tempHoming = TRUE) AND (_homingOld = FALSE) THEN
                // Rising edge on homing input
                _extendedCommand.%X2 := TRUE;
                IF FALSE
                    OR (config.homing.extendedMode = HOMING_ON_FIXED_STOP) // Extended Homing mode (active)
                    OR (config.homing.extendedMode = HOMING_ON_FIXED_STOP_WITH_MOVING_OUT_OF_CLAMPING)  // Extended Homing mode (active)
                    OR (config.homing.extendedMode = HOMING_ON_FIXED_STOP_WITH_MOVING_TO_TARGET_POSITION)
                    OR (config.homing.extendedMode = -1) AND ((config.homing.mode = ACTIVE_HOMING) OR (config.homing.mode = ACTIVE_HOMING_TO_DEF_VALUE)) // Extended Homing mode (active)
                THEN
                    // Active Homing selected
                    _basicCommand.%X10 := TRUE; // Cmd is BasicMotionCmd
                    _extendedCommand.%X2 := FALSE;
                    // ELSE
                    //   ; // Passive Homing selected
                    //   // Bit in extended cmd already written
                END_IF;

            ELSIF (tempHoming = FALSE) AND (_homingOld = TRUE) THEN
                // Falling edge on homing input
                _extendedCommand.%X2 := FALSE;
                _basicCommand.%X10 := FALSE;
                // ELSE
                //   ; // Do nothing - wait for rising / Falling edge
            END_IF;
            _basicCommand.%X7 := gearInRelative;
            _basicCommand.%X8 := gearInAbsolute;
            _basicCommand.%X12 := gearInVelocity;
            _basicCommand.%X9 := camIn;
            _basicCommand.%X11 := gearOutCamOut;
            _supImpCommand.%X1 := phasing;
            _supImpCommand.%X2 := offset;

            // Statemachine for synchronized motion simulation

            REPEAT
                tempStateChangeActive := FALSE;
                CASE _syncMotionSimulationState OF
                    AXIS_NOT_IN_SIM:
                        // Axis NOT in simulation
                        IF (config.power.syncMotionSimulation = TRUE) THEN
                            // SynchronizedMotionSimulation is set
                            IF (tempEnableAxis = FALSE) AND (_enableAxisOld = TRUE) THEN
                                // Falling edge at enableAxis --> set simulation
                                CASE config.power.syncMotionSimulationExtendedMode OF
                                    -1: // Automatic when axis is in synchronous operation
                                        IF tempStatusWord.%X22 THEN // Check if axis is in synchronous operation
                                            _syncMotionSimulationState := AXIS_STATE_SET_SIM;
                                            _enableAxis := TRUE;
                                            tempStateChangeActive := TRUE;
                                        ELSE
                                            _enableAxis := tempEnableAxis;
                                        END_IF;

                                    0: // Start always simulation
                                        _syncMotionSimulationState := AXIS_STATE_SET_SIM;
                                        _enableAxis := TRUE;
                                        tempStateChangeActive := TRUE;
                                ELSE
                                    _enableAxis := tempEnableAxis; // : disable axis anyway
                                    // Error - Invalid extended mode
                                    _status := AxisStatus#ERR_INVALID_SYNCHRONIZED_EXTENDED_MODE;
                                    _statusText := STRING#'ERR_INVALID_SYNCHRONIZED_EXTENDED_MODE';
                                    _errorAutoCleared := TRUE;
                                    _diagnostics.basicMotionState := _basicMotionState;
                                    _diagnostics.superimposedMotionState := _supImpMotionState;
                                    _diagnostics.subfunctionStatus := WORD#0000;
                                    _subfunctionStatus := AxisStatus#STATUS_NO_CALL;
                                END_CASE;
                            ELSE
                                // FALSE or rising edge at input enableAxis
                                _enableAxis := tempEnableAxis;
                            END_IF;
                        ELSE
                            // SynchronizedMotionSimulation not set
                            // MC_POWER is only controlled by enableAxis input
                            _enableAxis := tempEnableAxis;
                        END_IF;

                    AXIS_STATE_SET_SIM:
                        // Set the axis in simulation
                        //----------------------------------------------------------
                        // Enable SynchronizedMotionSimulation
                        _instSyncMotionSimulation(Slave := _refSyncAxis^,
                                                  Enable := TRUE);
                        //----------------------------------------------------------
                        IF (_instSyncMotionSimulation.InSimulation = TRUE) THEN
                            _enableAxis := FALSE;
                            // Axis in Simulation - Change state
                            _syncMotionSimulationState := AXIS_DISABLE;
                        ELSIF (_instSyncMotionSimulation.Error = TRUE) THEN
                            // Error occurred - Disable Axis immediately
                            _enableAxis := FALSE;
                            _syncMotionSimulationState := AXIS_STATE_RESET_SIM;
                        // ELSE
                            //   ; // Wait for Axis is in simulation
                        END_IF;

                    AXIS_DISABLE:
                        // Disable axis
                        //----------------------------------------------------------
                        // Enable SynchronizedMotionSimulation
                        _instSyncMotionSimulation(Slave := _refSyncAxis^,
                                                  Enable := TRUE);
                        //----------------------------------------------------------
                        IF (_instPower.Error = TRUE) THEN
                            _syncMotionSimulationState := AXIS_STATE_RESET_SIM;
                        ELSIF (_instPower.Status = FALSE) THEN
                            // Axis disabled
                            _syncMotionSimulationState := AXIS_STATE_IN_SIM;
                        // ELSE
                            //   ; // Wait for Axis is disabled
                        END_IF;

                    AXIS_STATE_IN_SIM:
                        // Axis is in simulation
                        //----------------------------------------------------------
                        // Enable SynchronizedMotionSimulation
                        _instSyncMotionSimulation(Slave := _refSyncAxis^,
                                                  Enable := TRUE);
                        //----------------------------------------------------------
                        IF (tempEnableAxis = TRUE) AND (_enableAxisOld = FALSE) THEN
                            // Rising edge at enableAxis --> reset simulation
                            _syncMotionSimulationState := AXIS_ENABLE;
                            _enableAxis := TRUE;
                            tempStateChangeActive := TRUE;
                        ELSIF (config.power.syncMotionSimulation = FALSE) THEN
                            // End of synchronizedMotionSimulation by config without starting Axis
                            _syncMotionSimulationState := AXIS_STATE_RESET_SIM;
                            tempStateChangeActive := TRUE;
                        // ELSE
                            //   ; // Wait for rising edge at enableAxis
                        END_IF;

                    AXIS_ENABLE:
                        // Enable Axis
                        //----------------------------------------------------------
                        // Enable SynchronizedMotionSimulation while axis is enabling
                        _instSyncMotionSimulation(Slave := _refSyncAxis^,
                                                  Enable := TRUE);
                        //----------------------------------------------------------

                        IF (tempEnableAxis = FALSE) AND (_enableAxisOld = TRUE) THEN
                            _syncMotionSimulationState := AXIS_STATE_RESET_SIM;
                            _enableAxis := FALSE;
                        ELSIF (tempStatusWord.%X0 = TRUE) OR (_instPower.Error = TRUE)
                        // Reset simulation if axis is enabled or MC_POWER.STATUS = FALSE (Axis Error)
                        THEN
                            // FALSE on enable input
                            _syncMotionSimulationState := AXIS_STATE_RESET_SIM;
                            tempStateChangeActive := TRUE;
                        // ELSE
                            //   ; // Wait for Axis is Enabled
                        END_IF;

                    AXIS_STATE_RESET_SIM:
                        // Reset the axis simulation
                        //----------------------------------------------------------
                        // Enable SynchronizedMotionSimulation
                        _instSyncMotionSimulation(Slave := _refSyncAxis^,
                                                Enable := FALSE);
                        //----------------------------------------------------------
                        IF (_instSyncMotionSimulation.InSimulation = FALSE) AND (_instSyncMotionSimulation.Busy = FALSE) THEN
                            // Axis simulation is disabled
                            _syncMotionSimulationState := AXIS_NOT_IN_SIM;
                        // ELSE
                            //   ; // Wait for axis simulation is disabled
                        END_IF;

                        IF (tempEnableAxis = FALSE) AND (_enableAxisOld = TRUE) THEN
                            _enableAxis := FALSE;
                        END_IF;
                ELSE
                    // Errorhandling
                    _status := AxisStatus#ERR_UNDEFINED_MOTION_SIMULATION_STATE;
                    _statusText := STRING#'ERR_UNDEFINED_MOTION_SIMULATION_STATE';
                    _errorUserCleared := TRUE;
                    _diagnostics.subfunctionStatus := WORD#0000;
                    _subfunctionStatus := AxisStatus#STATUS_NO_CALL;
                    _diagnostics.basicMotionState := _basicMotionState;
                    _diagnostics.superimposedMotionState := _supImpMotionState;
                    // Set error state
                    _state := FB_ERROR;
                END_CASE;
            UNTIL (tempStateChangeActive = FALSE)
            END_REPEAT;

            // Evaluation of MC_Command
            IF (_instSyncMotionSimulation.Error = TRUE) AND (_synchronizedMotionErrorOld = FALSE) THEN
                // Errorhandling - Set error only at rising edge
                _errorAutoCleared := TRUE;
                _status := AxisStatus#ERR_MC_SYNCHRONIZEDMOTIONSIMULATION;
                _statusText := STRING#'ERR_MC_SYNCHRONIZEDMOTIONSIMULATION';
                _diagnostics.basicMotionState := _basicMotionState;
                _diagnostics.superimposedMotionState := _supImpMotionState;
                _diagnostics.subfunctionStatus := _instSyncMotionSimulation.ErrorId;
                _subfunctionStatus := _instSyncMotionSimulation.ErrorId;
            ELSIF (_instSyncMotionSimulation.Error = FALSE) AND (_status = AxisStatus#ERR_MC_SYNCHRONIZEDMOTIONSIMULATION)
            THEN
                // Reset error if error gone at respective Status
                _errorAutoCleared := FALSE;
                _status := AxisStatus#STATUS_SUBSEQUENT_CALL;
                _statusText := STRING#'STATUS_SUBSEQUENT_CALL';
            END_IF;
            _synchronizedMotionErrorOld := _instSyncMotionSimulation.Error;
            tempEnableAxis := _enableAxis;

            // Enable and disable axis
            IF (config.power.externalMC_PowerCall = FALSE) THEN
                // Call MC_POWER
                // Do not call the MC_Power instance if the axis is successfully enabled -> Reduce the runtime of the LAxisCtrl block
                // Only call the instance if at least one of the following conditions is fulfilled
                IF ((tempEnableAxis = TRUE) AND ((_instPower.Busy = FALSE) OR (_instPower.Status = FALSE))) // "enable axis" is given and enabling via MC_Power is in progress
                    OR (tempStatusWord.%X0 = FALSE) // Axis is disabled
                    OR (tempEnableAxis = FALSE) // "Remove axis enable" is set
                    OR (_instPower.Error = TRUE) // An error occurred in Motion Control instruction "MC_Power"
                THEN // Call the MC_Power instance
                    _instPower(Axis := _refAxis^,
                               Enable := tempEnableAxis,
                               StartMode := config.power.startMode,
                               StopMode := config.power.stopMode);
                END_IF;

                // Set and Reset of Error
                IF (_instPower.Error = TRUE) AND
                    ((_status = AxisStatus#STATUS_SUBSEQUENT_CALL) OR (_powerErrorOld = FALSE))
                THEN
                    // Error is set at rising edge of MC_POWER.Error
                    // Errorhandling
                    _status := AxisStatus#ERR_MC_POWER;
                    _statusText := STRING#'ERR_MC_POWER';
                    _errorAutoCleared := TRUE;
                    _diagnostics.basicMotionState := _basicMotionState;
                    _diagnostics.superimposedMotionState := _supImpMotionState;
                    _diagnostics.subfunctionStatus := _instPower.ErrorId;
                    _subfunctionStatus := _instPower.ErrorId;

                ELSIF (_status = AxisStatus#ERR_MC_POWER) AND (_instPower.Error = FALSE)
                THEN
                    // Reset Error
                    _status := AxisStatus#STATUS_SUBSEQUENT_CALL;
                    _statusText := STRING#'STATUS_SUBSEQUENT_CALL';
                    _errorAutoCleared := FALSE;

                ELSIF (tempEnableAxis = TRUE) AND (_enableAxisOld = FALSE) THEN
                    // Reset Error
                    _status := AxisStatus#STATUS_SUBSEQUENT_CALL;
                    _statusText := STRING#'STATUS_SUBSEQUENT_CALL';
                    _errorAutoCleared := FALSE;
                    _diagnostics := _emptyDiagnostics;
                // ELSE
                    //   ; // Do nothing
                END_IF;
            END_IF;

            IF tempOpenBrake AND NOT _openBrakeOld THEN
                // Open
                _instSetAxisSTW(Axis := _refSpeedAxis^,
                                Execute := FALSE,
                                STW1 := MASK_STW_BIT12,
                                STW1BitMask := MASK_STW_BIT12);
                _brakeChangeActive := TRUE;
                _brakeOpened := TRUE;

            ELSIF NOT tempOpenBrake AND _openBrakeOld THEN
                // Close
                _instSetAxisSTW(Axis := _refSpeedAxis^,
                                Execute := FALSE,
                                STW1 := WORD#16#0000,
                                STW1BitMask := MASK_STW_BIT12);
                _brakeChangeActive := TRUE;
                _brakeOpened := FALSE;
            END_IF;

            IF _brakeChangeActive THEN
                // Call of MC command
                _instSetAxisSTW(Axis := _refSpeedAxis^,
                                Execute := TRUE);

                IF NOT _instSetAxisSTW.Busy THEN
                    _brakeChangeActive := FALSE;
                END_IF;
            END_IF;

            // Edge detection
            _openBrakeOld := tempOpenBrake;
        END_IF;

        //----------------------------------------------------------------------------------------------
        // Resolve TO reference of master and cam
        //----------------------------------------------------------------------------------------------
        // resolve reference for master input as TO_Axis (every synchronous operation needs at least a type of TO_Axis for its master input)
        IF master <> UINT#0 AND master <> _masterOld THEN
            _refMasterAxis := AsAxisRef(master);

            // TODO: generate other error for this case?
            IF _refMasterAxis = NULL THEN
                // Invalid axis
                error := TRUE;
                _errorUserCleared := TRUE;
                status := AxisStatus#ERR_INVALID_AXIS;
                statusText := STRING#'ERR_INVALID_AXIS';
                diagnostics.status := AxisStatus#ERR_INVALID_AXIS;
            END_IF;
        END_IF;

        _masterOld := master;

        // resolve reference for cam input as TO_CamBase (every cam operation needs at least a type of TO_CamBase for its cam input)
        IF cam <> UINT#0 AND cam <> _camOld THEN
            _refCamBase := AsCamBaseRef(cam);

            // TODO: generate other error for this case?
            IF _refCamBase = NULL THEN
                // Invalid axis
                error := TRUE;
                _errorUserCleared := TRUE;
                status := AxisStatus#ERR_INVALID_AXIS;
                statusText := STRING#'ERR_INVALID_AXIS';
                diagnostics.status := AxisStatus#ERR_INVALID_AXIS;
            END_IF;
        END_IF;

        _camOld := cam;

        //----------------------------------------------------------------------------------------------
        // FB Statemachine
        //----------------------------------------------------------------------------------------------
        CASE _state OF
            AXIS_MOTION:
                // Check command inputs
                IF (_extendedCommand = CMD_NO_SELECTION)
                    AND (_basicCommand = CMD_NO_SELECTION)
                    AND (_supImpCommand = CMD_NO_SELECTION)
                THEN
                    // Command is reset
                    IF (_instPower.Error = TRUE) THEN
                        // Errorhandling
                        _status := AxisStatus#ERR_MC_POWER;
                        _statusText := STRING#'ERR_MC_POWER';
                        _errorAutoCleared := TRUE;
                    ELSIF (_instSyncMotionSimulation.Error = TRUE) THEN
                        ; // Do nothing

                    ELSIF (_instTorqueLimiting.Error = TRUE) THEN
                        ; // Do not reset if torque limiting error is pending

                    ELSE
                        // Reset Error only if no Error at MC_POWER is present
                        _status := AxisStatus#STATUS_SUBSEQUENT_CALL;
                        _statusText := STRING#'STATUS_SUBSEQUENT_CALL';
                        _errorAutoCleared := FALSE;
                    END_IF;

                ELSIF (_extendedCommand = _extendedCommandOld)
                    AND (_basicCommand = _basicCommandOld)
                    AND (_supImpCommand = _supImpCommandOld)
                THEN
                    ; // No change at command - do nothing

                ELSE
                    // Command changed
                    tempNewExtendedCmd := NO_SELECTION;
                    tempNewBasicMotionCmd := NO_SELECTION;
                    tempNewSupImpCmd := NO_SELECTION;
                    tempErrorInCmd := FALSE;

                    // Check basic motion command
                    IF (_basicCommand = _basicCommandOld) THEN
                        ; // Do nothing
                    ELSE
                        // Evaluate rising edges for basic motion command word - all rising edges of basic command word saved in tempRisingBasicCmd
                        tempRisingCmd := ((_basicCommand XOR _basicCommandOld) AND _basicCommand);
                        tempCountRisEdges := USINT#0; // Initialize counter for rising edges
                        // Count rising edges in tempRisingBasicCmd
                        FOR tempIndex := BITPOSITION_BASIC_MOTION_CMD TO BIT_POS_LAST DO
                            tempDword := SHR(tempRisingCmd, TO_USINT(tempIndex));
                            // Check for rising edge
                            IF (tempDword.%X0 = TRUE) THEN
                                tempCountRisEdges := tempCountRisEdges + USINT#1; // Increment at rising edge
                            END_IF;
                        END_FOR;
                        IF (tempRisingCmd.%X2 = TRUE) OR (tempRisingCmd.%X3 = TRUE) THEN
                            tempCountRisEdges := tempCountRisEdges + USINT#1; // jogForward AND/OR jogBackward is standing for 1 Command/rising edge
                        END_IF;

                        // Check Basic motion command
                        IF (tempCountRisEdges = 1)
                            OR (tempRisingCmd.%X0 = TRUE) // fastStop selected
                            OR (tempRisingCmd.%X1 = TRUE) // Stop selected
                        THEN
                            // Valid basic motion command selected
                            IF (tempRisingCmd.%X0 = TRUE) THEN
                                // FastStop selected
                                _state := AXIS_FAST_STOPPING;
                                tempNewBasicMotionCmd := FAST_STOP_SELECTED;
                                tempStopCmdSelected := TRUE;
                            ELSIF (tempRisingCmd.%X1 = TRUE) THEN
                                // Stop selected
                                tempNewBasicMotionCmd := STOP_SELECTED;
                                tempStopCmdSelected := TRUE;
                            ELSE
                                // Valid basic command priority 3 selected
                                // Set basic motion state
                                tempNewBasicMotionCmd := TO_DINT(tempRisingCmd);
                            END_IF;

                        ELSIF (tempCountRisEdges > 1) THEN
                            // Errorhandling - Invalid command
                            _status := AxisStatus#ERR_INVALID_BASIC_MOTION_CMD;
                            _statusText := STRING#'ERR_INVALID_BASIC_MOTION_CMD';
                            tempErrorInCmd := TRUE;
                        // ELSE
                            //   ; // Falling edge detection
                        END_IF;
                    END_IF;

                    // Check superimposed motion command
                    IF (_supImpCommand = _supImpCommandOld) THEN
                        ; // Do nothing
                    ELSE
                        // Superimposed motion command selected
                        IF (tempErrorInCmd = FALSE) AND // No Stop command selected in current cycle
                            (tempStopCmdSelected = FALSE)
                        THEN
                            tempRisingCmd := ((_supImpCommand XOR _supImpCommandOld) AND _supImpCommand);
                            tempCountRisEdges := USINT#0; // Initialize counter for rising edges
                            // Count rising edges in tempRisingSupImpCmd
                            FOR tempIndex := BITPOSITION_SUPERIMPOSED_MOTION_CMD TO BIT_POS_LAST DO
                                tempDword := SHR(tempRisingCmd, TO_USINT(tempIndex));
                                // Check for rising edge
                                IF (tempDword.%X0 = TRUE) THEN
                                    tempCountRisEdges := tempCountRisEdges + USINT#1;
                                END_IF;
                            END_FOR;

                            IF (tempCountRisEdges = 1) THEN
                                // Valid superimposed motion command
                                tempNewSupImpCmd := TO_DINT(tempRisingCmd);

                            ELSIF (tempCountRisEdges > 1) THEN
                                // Invalid Superimposed motion command
                                _status := AxisStatus#ERR_INVALID_SUPERIMPOSED_MOTION_CMD;
                                _statusText := STRING#'ERR_INVALID_SUPERIMPOSED_MOTION_CMD';
                                tempErrorInCmd := TRUE;
                            // ELSE
                                //   ; // Falling edge detection
                            END_IF;
                        // ELSE
                            //   ; // Stop or Faststop command selected OR error in BasicCommand
                        END_IF;
                    END_IF;

                    // Check extended command (reset, homing, torquelimiting)
                    IF (_extendedCommand = _extendedCommandOld) THEN
                        ; // Do nothing
                    ELSE
                        // Extended command selected
                        IF (tempErrorInCmd = FALSE) THEN
                            tempRisingCmd := ((_extendedCommand XOR _extendedCommandOld) AND _extendedCommand);
                            // Rising edge on torquelimiting command
                            IF (tempRisingCmd.%X1 = TRUE) THEN
                                tempNewExtendedCmd.%X1 := TRUE;
                                // Rising Edge at Homing on Fixed Stop and Torquelimiting
                                IF (tempNewBasicMotionCmd.%X10 = TRUE) AND (config.homing.extendedMode = 0) THEN
                                    // Errorhandling
                                    _status := AxisStatus#ERR_INVALID_EXTENDED_CMD;
                                    _statusText := STRING#'ERR_INVALID_EXTENDED_CMD';
                                    tempErrorInCmd := TRUE;
                                    tempNewExtendedCmd.%X1 := FALSE;

                                ELSIF (_torqueLimitingState = FIXED_STOP_DETECTION_ACTIVE)
                                THEN
                                    // Torquelimiting rejected because MC_TorqueLimiting is used during homing on fixed stop functionality
                                    _status := AxisStatus#ERR_TORQUE_LIMITING_NOT_ALLOWED;
                                    _statusText := STRING#'ERR_TORQUE_LIMITING_NOT_ALLOWED';
                                    tempErrorInCmd := TRUE;
                                    tempNewExtendedCmd.%X1 := FALSE;
                                    // ELSE
                                    //   ; // Start torquelimiting functionality
                                END_IF;
                            END_IF;

                            // Rising edge on passive homing command
                            IF (tempRisingCmd.%X2 = TRUE) THEN
                                tempNewExtendedCmd.%X2 := TRUE;
                                IF TRUE
                                    AND (_basicMotionState = ACTIVE_HOMING_SELECTED)
                                    AND ((_activeHomingState = HOMING_ON_FIXED_STOP) OR (_activeHomingState = HOMING_ON_FIXED_STOP_WITH_MOVING_OUT_OF_CLAMPING) OR (_activeHomingState = HOMING_ON_FIXED_STOP_WITH_MOVING_TO_TARGET_POSITION))
                                    AND (_exeOfBasicMotion = CMD_BUSY)
                                THEN
                                    // Passive Homing selected at homing on fixed stop
                                    _status := AxisStatus#ERR_HOMING_MODE_NOT_ALLOWED;
                                    _statusText := STRING#'ERR_HOMING_MODE_NOT_ALLOWED';
                                    tempErrorInCmd := TRUE;
                                    tempNewExtendedCmd.%X2 := FALSE;
                                    // ELSE
                                    //   ; // No error occurred
                                END_IF;
                            END_IF;
                        ELSE
                            ; // Error in basic motion command or superimposed motion command
                        END_IF;
                    END_IF;

                    // Enable commands
                    IF (tempErrorInCmd = TRUE) AND (tempStopCmdSelected = FALSE) THEN
                        // Error in current command - No Execution
                        _errorAutoCleared := TRUE;
                        _diagnostics.subfunctionStatus := WORD#0000;
                        _subfunctionStatus := AxisStatus#STATUS_NO_CALL;
                        // Write diagnostics
                        _diagnostics.basicMotionState := _basicMotionState;
                        _diagnostics.superimposedMotionState := _supImpMotionState;
                        _resetIncJog := TRUE;
                        // Set next state
                        _state := AXIS_STOP_ON_ERROR_SELECTION;
                    ELSE
                        // No Error in command occurred
                        IF (
                            (tempNewExtendedCmd <> NO_SELECTION)
                            OR (tempNewBasicMotionCmd <> NO_SELECTION)
                            OR (tempNewSupImpCmd <> NO_SELECTION)
                            )
                            OR (tempStopCmdSelected = TRUE)
                        THEN

                            // New valid command selected
                            // Basic motion commands
                            IF (tempNewBasicMotionCmd <> NO_SELECTION) THEN
                                _mainSelectionState := CALL_BASIC_MOTION;

                                IF config.generalSettings.abortWaitingSyncCmd THEN
                                    // Get axis waiting function state
                                    IF (_typeAxis = SYNC_AXIS) THEN
                                        _waitingFunctionStateAbortAutomatic := _refSyncAxis^.StatusSynchronizedMotion.WaitingFunctionState;
                                    END_IF;

                                    CASE _waitingFunctionStateAbortAutomatic OF
                                        WFS_FS_GEARINPOS, // Waiting
                                        WFS_FS_CAMIN: // Waiting
                                            // Waiting sync command
                                            CASE tempNewBasicMotionCmd OF
                                                GEAR_IN_ABSOLUTE_SELECTED,
                                                GEAR_IN_VELOCITY_SELECTED,
                                                CAM_IN_SELECTED,
                                                GEAR_IN_RELATIVE_SELECTED,
                                                GEAR_OUT_CAM_OUT_SELECTED:
                                                    ; // New command aborts waiting sync command
                                            ELSE
                                                _mainSelectionState := ABORT_WAITING_GEARINPOS_OR_CAMIN; // Reset waiting absolute gearing / camIn command
                                            END_CASE;
                                    ELSE
                                        ;
                                    END_CASE;

                                    IF (_mainSelectionState = ABORT_WAITING_GEARINPOS_OR_CAMIN) THEN
                                        // Reset instance of MC_GearOut / MC_CamOut
                                        CASE _waitingFunctionStateAbortAutomatic OF
                                            WFS_FS_GEARINPOS: // Waiting
                                                _instGearOut(Slave := _refSyncAxis^,
                                                            Execute := FALSE,
                                                            SyncProfileReference := CANCEL_ONLY_WAITING_GEARING_CAMMING); // 5 = Abort waiting camming / gearing

                                            WFS_FS_CAMIN: // Waiting
                                                _instCamOut(Slave := _refSyncAxis^,
                                                            Execute := FALSE,
                                                            SyncProfileReference := CANCEL_ONLY_WAITING_GEARING_CAMMING); // 5 = Abort waiting camming / gearing
                                        END_CASE;
                                    END_IF;
                                ELSE
                                    // Automatic abort of waiting sync commands not enabled
                                    _waitingFunctionStateAbortAutomatic := -1;
                                END_IF;

                                _firstCycleBasicMotion := TRUE;
                                // Evaluate if Jog command is set
                                IF (tempNewBasicMotionCmd.%X2 = TRUE) OR (tempNewBasicMotionCmd.%X3 = TRUE) THEN
                                    _exeOfBasicMotion := CMD_BUSY;
                                    // Select Jogmode
                                    IF ((_basicCommand.%X2 = FALSE) AND (tempNewBasicMotionCmd.%X3 = TRUE)) OR // Rising edge at JogBackward and JogForward = FALSE
                                        ((_basicCommand.%X3 = FALSE) AND (tempNewBasicMotionCmd.%X2 = TRUE)) OR // Only rising edge at JogForward and JogBackward = FALSE
                                        ((tempNewBasicMotionCmd.%X2 = TRUE) AND (tempNewBasicMotionCmd.%X3 = TRUE)) // Rising edge at FW and BW
                                    THEN
                                        // One Input direction = False, other is rising edge, or both rising edge --> Start jog
                                        IF (_jogMode <> config.jog.mode) THEN
                                            _resetIncJog := TRUE;
                                        END_IF;
                                        _jogMode := config.jog.mode;
                                    ELSE
                                        // Rising edge at one input, the other is already TRUE - Dont Change Jogmode
                                        IF ((_basicMotionState = JOG_BACKWARD_SELECTED) OR (_basicMotionState = JOG_FORWARD_SELECTED)) AND (_jogMode <> JOG_MODE_CONTINUOUS)
                                        THEN
                                            _firstCycleBasicMotion := FALSE;
                                        END_IF;
                                    END_IF;
                                ELSE
                                    ; // Reset jog increment if other command than jog selected
                                    _resetIncJog := TRUE;
                                END_IF;

                                // Set new basic motion state
                                _basicMotionState := tempNewBasicMotionCmd;
                            END_IF;

                            // Superimposed motion commands
                            IF (tempNewSupImpCmd <> NO_SELECTION) THEN
                                _supImpMotionState := tempNewSupImpCmd;
                                _firstCycleSupImpMotion := TRUE;
                                _resetIncJog := TRUE;
                            END_IF;

                            // Extended commands

                            IF (tempNewExtendedCmd <> NO_SELECTION) THEN
                                IF (tempNewExtendedCmd.%X1 = TRUE) THEN
                                    // Rising edge on torquelimiting command
                                    IF (_torqueLimitingState = NO_TORQUE_LIMITING_ACTIVE) THEN
                                        // No torquelimiting active --> Enable torquelimiting
                                        _torqueLimitingState := TORQUE_LIMITING_SELECTED;
                                    END_IF;
                                END_IF;
                                // Homing command
                                IF (tempNewExtendedCmd.%X2 = TRUE) THEN
                                    _passiveHomingState := config.homing.extendedMode;
                                    _firstCycleHoming := TRUE;
                                    _resetIncJog := TRUE;
                                END_IF;
                            END_IF;

                        // Reset error
                        _status := AxisStatus#STATUS_SUBSEQUENT_CALL;
                        _statusText := STRING#'STATUS_SUBSEQUENT_CALL';
                        _errorAutoCleared := FALSE;
                        _diagnostics := _emptyDiagnostics;
                    // ELSE
                        //   ; // No rising edge at commands
                        END_IF;
                    END_IF;
                END_IF;

            AXIS_FAST_STOPPING:
                IF (config.fastStop.replaceStopPossible = FALSE) THEN
                    ; // Fast stop command can not be interrupted by another command
                    // State change is executed in FastStop implementation if command finished
                ELSE
                    _state := AXIS_MOTION;
                END_IF;

            AXIS_STOP_ON_ERROR_SELECTION,
            AXIS_STOP_ON_ERROR_EXECUTION:
                ; // Wait for stopping axis if StopOnError is configured
            FB_ERROR: // Error state
                ; // Do nothing, status already set

        ELSE
            // Errorhandling
            _status := AxisStatus#ERR_UNDEFINED_FB_STATE;
            _statusText := STRING#'ERR_UNDEFINED_FB_STATE';
            _errorUserCleared := TRUE;
            _diagnostics.subfunctionStatus := WORD#0000;
            _subfunctionStatus := AxisStatus#STATUS_NO_CALL;
            _diagnostics.basicMotionState := _basicMotionState;
            _diagnostics.superimposedMotionState := _supImpMotionState;
            // Set error state
            _state := FB_ERROR;
        END_CASE;

        //----------------------------------------------------------------------------------------------
        // Execution of reset functionality
        //----------------------------------------------------------------------------------------------

        // Firstcycle of command
        IF (_extendedCommand.%X0 = TRUE) AND (_extendedCommandOld.%X0 = FALSE) THEN
            _firstCycleReset := TRUE;
            // Reset MC_RESET command
            _instReset(Axis := _refAxis^,
                       Execute := FALSE,
                       Restart := config.generalSettings.resetWithRestart);
            _firstCycleResetError := FALSE;
            _resetState := CMD_BUSY;
        END_IF;

        CASE _resetState OF
            CMD_IDLE:
                ; // Do nothing

            CMD_BUSY:
                // Call MC_Command
                _instReset(Axis := _refAxis^,
                           Execute := _extendedCommand.%X0);

                // Evaluate MC_Command
                IF (_instReset.Error = TRUE) THEN
                    // Errorhandling
                    IF (_firstCycleResetError = FALSE) THEN
                        _errorAutoCleared := TRUE;
                        _status := AxisStatus#ERR_MC_RESET;
                        _statusText := STRING#'ERR_MC_RESET';
                        _diagnostics.basicMotionState := _basicMotionState;
                        _diagnostics.superimposedMotionState := _supImpMotionState;
                        _diagnostics.subfunctionStatus := _instReset.ErrorId;
                        _subfunctionStatus := _instReset.ErrorId;
                        _firstCycleResetError := TRUE;
                        // Set next state
                        _resetState := CMD_IDLE;
                        IF (_state = AXIS_MOTION) THEN
                        // Set TO_STOP_ON_ERROR State only if the current state is TO_MOTION
                        _state := AXIS_STOP_ON_ERROR_SELECTION;
                        END_IF;
                    END_IF;

                ELSIF (_instReset.Busy = FALSE) THEN
                    // Set next state
                    _resetState := CMD_IDLE;
                // ELSE
                //   ; // Command selected
                END_IF;
        ELSE
            // Errorhandling
            _status := AxisStatus#ERR_UNDEFINED_RESET_STATE;
            _statusText := STRING#'ERR_UNDEFINED_RESET_STATE';
            _errorUserCleared := TRUE;
            _diagnostics.subfunctionStatus := WORD#0000;
            _subfunctionStatus := AxisStatus#STATUS_NO_CALL;
            _diagnostics.basicMotionState := _basicMotionState;
            _diagnostics.superimposedMotionState := _supImpMotionState;
        END_CASE;

        //----------------------------------------------------------------------------------------------
        // Execution of functionalities of basic coordinate system
        //----------------------------------------------------------------------------------------------

        // Write diagnostics
        _diagnostics.basicMotionState := _basicMotionState;
        _diagnostics.superimposedMotionState := _supImpMotionState;
        REPEAT
            tempStateChangeActive := FALSE;
            // Statemachine for main selection state
            CASE _mainSelectionState OF
                CALL_BASIC_MOTION:
                    CASE _basicMotionState OF
                        NO_SELECTION:
                            ; // No execution

                        FAST_STOP_SELECTED:
                            ; // Implementation at end of code

                        STOP_SELECTED:
                            // No additional features

                            // Firstcycle of command
                            IF (_firstCycleBasicMotion = TRUE) THEN
                                // Reset HALT command
                                _instHalt(Axis := _refSpeedAxis^,
                                          Execute := FALSE,
                                          Deceleration := config.stop.deceleration,
                                          AbortAcceleration := config.stop.abortAcceleration,
                                          Jerk := config.stop.jerk,
                                          Mode := config.stop.haltMode); // New input 'Mode' as of Motion Control V9.0
                            END_IF;

                            // Call MC_Command
                            _instHalt(Axis := _refSpeedAxis^,
                                      Execute := _basicCommand.%X1 OR _firstCycleBasicMotion);

                            // Evaluate MC_Command
                            IF (_instHalt.Busy = FALSE) AND
                                (_instHalt.Error = FALSE) AND
                                (_instHalt.Done = FALSE) AND
                                (_instHalt.CommandAborted = FALSE)
                            THEN
                                // Return to NO_SELECTION if command finished
                                _basicMotionState := NO_SELECTION;

                            ELSIF (_instHalt.Error = TRUE) THEN
                                // Errorhandling
                                _status := AxisStatus#ERR_MC_HALT;
                                _statusText := STRING#'ERR_MC_HALT';
                                _errorAutoCleared := TRUE;
                                _diagnostics.subfunctionStatus := _instHalt.ErrorId;
                                _subfunctionStatus := _instHalt.ErrorId;
                                // Set next state
                                _state := AXIS_STOP_ON_ERROR_SELECTION;
                                _basicMotionState := NO_SELECTION;
                            // ELSE
                                //   ; // Command selected
                            END_IF;
